Universal Robots PolyScope program: Try1.urp

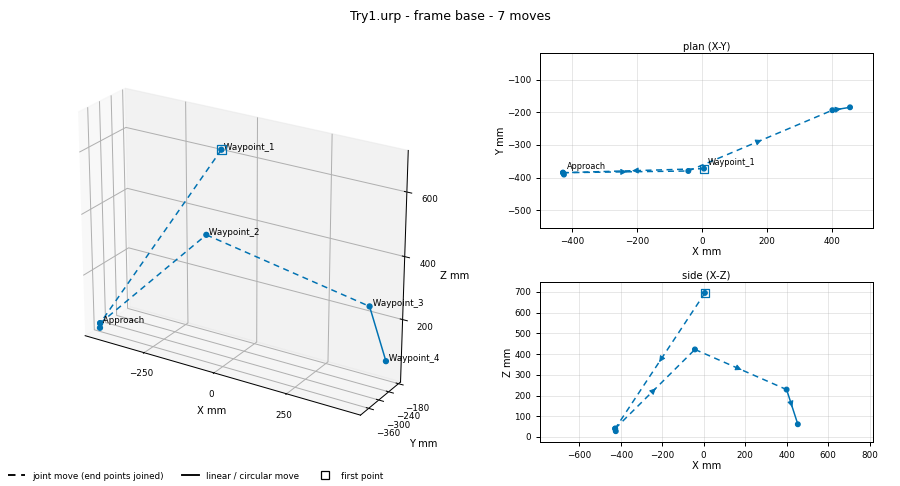
[picture p0: tool path of Try1.urp in frame base, 7 of 7 moves have a stored position in this frame; points joined in program order, loops and branches not executed]
Program Try1 (installation=default directory=/programs createdIn=5.14.5 lastSavedIn=5.14.5 robotSerialNumber=20195300809)
Calibrated DH parameters: a=[-0.000085, -0.20076, -0.212369, 0.000121, -0.000118, 0]; d=[0.15185, -26.306375, 24.753047, 1.684739, 0.085386, 0.092088]; alpha=[1.572149, -0.00522, -0.011864, 1.571339, -1.571085, 0]; deltaTheta=[0, 0.599885, -0.513355, -0.086555, 0.000006, 0]
InitVariablesNode variables(variable(name=Pallet_1_cnt_1, expression=1), variable(name=Pallet_1_lct, expression=1), variable(name=Pallet_1_lno, expression=1), variable(name=Pallet_1_sep, expression=False), variable(name=Pallet_1_tct, expression=1))
Robot Program (runOnlyOnce=true)
  MoveJ speed 60 deg/s, acceleration 80 deg/s^2 (useActiveTCP=true) feature=Base
    Waypoint Waypoint_1: TCP in base x=5.945 y=-372.701 z=694.671 mm, rx=-0.0179 ry=2.2102 rz=-2.2166 rad; joints [-0.001, -90.003, 0.003, -89.999, -0.001, -0.002] deg; TCP offset x=0 y=0 z=150 mm, rx=0 ry=0 rz=0 rad
  URCap Palletizing (polyscope-pallet-impl, Universal Robots) dataModel(palletFeature=Base, isPalletizing=false, Variable(key=name, variable(name=Pallet_1)), Variable(key=globalCountingVariable, variable(name=Pallet_1_cnt_1, initializeExpression=1)), Variable(key=layerNumberVariable, variable(name=Pallet_1_lno, initializeExpression=1)), Variable(key=layerCountingVariable, variable(name=Pallet_1_lct, initializeExpression=1)), Variable(key=handleSeparatorVariable, variable(name=Pallet_1_sep, initializeExpression=False)), Variable(key=totalCountVariable, variable(name=Pallet_1_tct, initializeExpression=1)), Length(key=objectHeight value=0.05 unit=M), Variable(key=referencePoint, variable(featureName=referencePoint)), Variable(key=separatorPoint, variable(featureName=separatorPoint))); state(isChildrenLocked=true)
    URCap Patterns (polyscope-pallet-impl, Universal Robots) state(isChildrenLocked=true)
      URCap Pattern (polyscope-pallet-impl, Universal Robots) dataModel(UUID=7f3fea2c-f655-493e-9669-857d3912d49b, patternType=IRREGULAR, Variable(key=nameVariable, variable(name=Irreg_Pattern_1))); state(isChildrenLocked=true)
        URCap Item (polyscope-pallet-impl, Universal Robots) dataModel(UUID=a94b10b2-0e9c-4eb9-b82d-31559a1a1133, patternType=IRREGULAR, index=0, calibrationDeltaTheta=[2.0871938292282843E-8, 0.5998849625986696, -0.513354759222901, -0.08655474087847535, 6.239817607139875E-6, -6.658617090343766E-8], calibrationA=[-8.52060452638757E-5, -0.2007601879611388, -0.2123691625519033, 1.2105607098011576E-4, -1.1833705743435544E-4, 0.0], calibrationD=[0.15184970286177432, -26.306374840159272, 24.75304670983349, 1.6847390881089916, 0.085385969004481, 0.09208826337351553], calibrationAlpha=[1.5721487795181908, -0.005219907129425837, -0.011864150755780208, 1.5713392161993658, -1.5710853432049288, 0.0], calibrationJointChecksum=[-1860213401, -1859864814, -1494669377, -1328152407, -1329437658, -1329056899], calibrationStatus=2, calibrationValidChecksum=true, baseToFeature=[0.0, 0.0, 0.0, 0.0, 0.0, 0.0], TCPOffset=[-5.976879858260453E-7, 9.740547549541567E-6, 0.15001564745172993, -3.112409760540105E-5, -2.3606128628809766E-5, 3.04322234517268E-5], Variable(key=variable, variable(name=Item_1)), JointPositions(key=jointpositions, JointPosition(key=[1], Angle(key=pos value=0.444656 unit=RAD)), JointPosition(key=[2], Angle(key=pos value=-0.520606 unit=RAD)), JointPosition(key=[3], Angle(key=pos value=0.585085 unit=RAD)), JointPosition(key=[4], Angle(key=pos value=-1.814807 unit=RAD)), JointPosition(key=[5], Angle(key=pos value=-1.447447 unit=RAD)), JointPosition(key=[6], Angle(key=pos value=-1.023818 unit=RAD))))
    URCap Layers (polyscope-pallet-impl, Universal Robots) dataModel(separators=[false], selectedPatterns=[7f3fea2c-f655-493e-9669-857d3912d49b])
    URCap At Each Item (polyscope-pallet-impl, Universal Robots) dataModel(selectedPattern=7f3fea2c-f655-493e-9669-857d3912d49b, selectedPosition=a94b10b2-0e9c-4eb9-b82d-31559a1a1133, Approach_calibrationDeltaTheta=[2.0871938292282843E-8, 0.5998849625986696, -0.513354759222901, -0.08655474087847535, 6.239817607139875E-6, -6.658617090343766E-8], Approach_calibrationA=[-8.52060452638757E-5, -0.2007601879611388, -0.2123691625519033, 1.2105607098011576E-4, -1.1833705743435544E-4, 0.0], Approach_calibrationD=[0.15184970286177432, -26.306374840159272, 24.75304670983349, 1.6847390881089916, 0.085385969004481, 0.09208826337351553], Approach_calibrationAlpha=[1.5721487795181908, -0.005219907129425837, -0.011864150755780208, 1.5713392161993658, -1.5710853432049288, 0.0], Approach_calibrationJointChecksum=[-1860213401, -1859864814, -1494669377, -1328152407, -1329437658, -1329056899], Approach_calibrationStatus=2, Approach_calibrationValidChecksum=true, Approach_baseToFeature=[0.0, 0.0, 0.0, 0.0, 0.0, 0.0], Approach_TCPOffset=[-1.1231275834290075E-5, 1.829168926326119E-7, 0.15000021294691582, -4.888694274368382E-7, -1.2062663179163743E-5, -2.9953026467210174E-5], Exit_calibrationDeltaTheta=[2.0871938292282843E-8, 0.5998849625986696, -0.513354759222901, -0.08655474087847535, 6.239817607139875E-6, -6.658617090343766E-8], Exit_calibrationA=[-8.52060452638757E-5, -0.2007601879611388, -0.2123691625519033, 1.2105607098011576E-4, -1.1833705743435544E-4, 0.0], Exit_calibrationD=[0.15184970286177432, -26.306374840159272, 24.75304670983349, 1.6847390881089916, 0.085385969004481, 0.09208826337351553], Exit_calibrationAlpha=[1.5721487795181908, -0.005219907129425837, -0.011864150755780208, 1.5713392161993658, -1.5710853432049288, 0.0], Exit_calibrationJointChecksum=[-1860213401, -1859864814, -1494669377, -1328152407, -1329437658, -1329056899], Exit_calibrationStatus=2, Exit_calibrationValidChecksum=true, Exit_baseToFeature=[0.0, 0.0, 0.0, 0.0, 0.0, 0.0], Exit_TCPOffset=[7.7050607285023E-6, 2.877704777926038E-5, 0.15002425182997436, -1.2671802509042467E-4, -1.1709091599254946E-5, 3.160996968116104E-5], currentWizardState=SHOW_DONE, Pose(key=refBaseToFeature, Position(key=posePosition, Length(key=X value=0 unit=M), Length(key=Y value=0 unit=M), Length(key=Z value=0 unit=M)), Rotation(key=poseRotation, Angle(key=RX value=0 unit=RAD), Angle(key=RY value=0 unit=RAD), Angle(key=RZ value=0 unit=RAD))), Pose(key=refPose, Position(key=posePosition, Length(key=X value=-0.423915 unit=M), Length(key=Y value=-0.39092 unit=M), Length(key=Z value=0.027871 unit=M)), Rotation(key=poseRotation, Angle(key=RX value=-0.092889 unit=RAD), Angle(key=RY value=-3.016827 unit=RAD), Angle(key=RZ value=0.294491 unit=RAD))), JointPositions(key=Approach_jointpositions, JointPosition(key=[1], Angle(key=pos value=0 unit=RAD)), JointPosition(key=[2], Angle(key=pos value=-1.570796 unit=RAD)), JointPosition(key=[3], Angle(key=pos value=0 unit=RAD)), JointPosition(key=[4], Angle(key=pos value=-1.570796 unit=RAD)), JointPosition(key=[5], Angle(key=pos value=0 unit=RAD)), JointPosition(key=[6], Angle(key=pos value=0 unit=RAD))), JointPositions(key=Exit_jointpositions, JointPosition(key=[1], Angle(key=pos value=2.608497 unit=RAD)), JointPosition(key=[2], Angle(key=pos value=-0.427014 unit=RAD)), JointPosition(key=[3], Angle(key=pos value=0.015077 unit=RAD)), JointPosition(key=[4], Angle(key=pos value=-1.199585 unit=RAD)), JointPosition(key=[5], Angle(key=pos value=-1.519749 unit=RAD)), JointPosition(key=[6], Angle(key=pos value=-0.613197 unit=RAD))))
      URCap Generated Movements (polyscope-pallet-impl, Universal Robots) state(isChildrenLocked=true)
        MoveJ speed 60 deg/s, acceleration 80 deg/s^2 (useActiveTCP=true) feature=referencePoint
          Waypoint Approach: TCP in base x=-426.869 y=-385.161 z=40.348 mm, rx=-0.1445 ry=-3.0302 rz=0.3154 rad; joints [25.477, -29.826, 33.526, -103.98, -82.931, -58.66] deg; feature pose in base x=-423.915 y=-390.92 z=27.871 mm, rx=-0.0929 ry=-3.0168 rz=0.2945 rad
        MoveL speed 250 mm/s, acceleration 1200 mm/s^2 (useActiveTCP=true) feature(featureName=referencePoint)
          Waypoint ToolActionPoint: TCP in base x=-423.915 y=-390.92 z=27.871 mm, rx=-0.0929 ry=-3.0168 rz=0.2945 rad; joints [26.654, -28.975, 35.357, -107.206, -84.067, -59.536] deg; TCP offset x=0.019 y=-0.006 z=149.979 mm, rx=0 ry=0 rz=0.0001 rad
        Folder Tool action
          URCap Gripper Activate (Robotiq_Grippers, Robotiq Inc.) dataModel(ResetAndActivateKey=false)
          URCap Gripper (Robotiq_Grippers, Robotiq Inc.) dataModel(position=100.0, force=100.0, speed=100.0, positionInDouble=100.0, forceInDouble=100.0, speedInDouble=100.0, slaveIds=[3], blocking=true)
        MoveL speed 250 mm/s, acceleration 1200 mm/s^2 (useActiveTCP=true) feature(featureName=referencePoint)
          Waypoint Approach: TCP in base x=-426.869 y=-385.161 z=40.348 mm, rx=-0.1445 ry=-3.0302 rz=0.3154 rad; joints [25.477, -29.826, 33.526, -103.98, -82.931, -58.66] deg; TCP offset x=0 y=0 z=150 mm, rx=0 ry=0 rz=0 rad
  MoveJ speed 60 deg/s, acceleration 80 deg/s^2 (useActiveTCP=true) feature=Base
    Waypoint Waypoint_2: TCP in base x=-42.208 y=-379.929 z=422.184 mm, rx=-0.0748 ry=-2.9117 rz=0.8251 rad; joints [56.009, -76.241, 10.628, -55.071, -79.952, -27.653] deg
  MoveJ speed 60 deg/s, acceleration 80 deg/s^2 (useActiveTCP=true) feature=Base
    Waypoint Waypoint_3: TCP in base x=399.86 y=-193.404 z=228.673 mm, rx=2.2461 ry=-2.0976 rz=0.1728 rad; joints [139.128, -57.618, 29.531, -68.211, -94.731, -44.742] deg
  MoveL speed 250 mm/s, acceleration 1200 mm/s^2 (useActiveTCP=true) feature=Base
    Waypoint Waypoint_4: TCP in base x=454.09 y=-184.487 z=61.293 mm, rx=2.1868 ry=-2.2038 rz=-0.0273 rad; joints [143.334, -41.748, 44.606, -91.566, -92.83, -36.267] deg
  URCap Gripper (Robotiq_Grippers, Robotiq Inc.) dataModel(position=0.0, force=100.0, speed=100.0, positionInDouble=0.0, forceInDouble=100.0, speedInDouble=100.0, slaveIds=[3], blocking=true)
